PROGRAM PRG_Methods
VAR
END_VAR

GVL_methods.Job(); // Cyclic execution of function block that is exposed as "job method"

END_PROGRAM

(* stored: Version 1.1.0.1
   POU PRG_Methods: Id {9ef9c5cc-c02c-44d8-bf7a-ae8e462a8731}, SpecialFunc None *)
